// SIMATIC STEP 7 (V5.x) project aplicaciopnes
// CPU: CPU 314C-2 DP
// CPU: CPU 314C-2 DP
// CPU: CPU 314C-2 DP
// CPU: CPU 314C-2 DP
// CPU: CPU 314C-2 DP
// CPU: CPU 314C-2 DP
// CPU: CPU 314C-2 DP
// station: Hardware
// station: secuencial
// station: P_ADR_BUS
// station: Hardware
// station: motores secuenciales
// station: P_ADR_BUS
// station: Hardware
// station: mot sec original
// station: P_ADR_BUS
// station: Hardware
// station: agitador con agua
// station: P_ADR_BUS
// station: Hardware
// station: bombas con una lampara
// station: P_ADR_BUS
// station: Hardware
// station: funciones
// station: P_ADR_BUS
// station: Hardware
// station: tres tanques llenado sec
// station: P_ADR_BUS
// program: Programa S7(1)
// program: Programa S7(2)
// program: Programa S7(3)
// program: Programa S7(5)
// program: Programa S7(6)
// program: Programa S7(7)
// program: Programa S7(8)

SYMBOL_TABLE
"arranque"	I 124.0	BOOL
"paro"	I 124.1	BOOL
"L1"	Q 124.0	BOOL
"L2"	Q 124.1	BOOL
"L3"	Q 124.2	BOOL
END_SYMBOL_TABLE

ORGANIZATION_BLOCK OB 1
TITLE = "Main Program Sweep (Cycle)"
VERSION : 0.1
VAR_TEMP
  OB1_EV_CLASS : BYTE ;	//Bits 0-3 = 1 (Coming event), Bits 4-7 = 1 (Event class 1)
  OB1_SCAN_1 : BYTE ;	//1 (Cold restart scan 1 of OB 1), 3 (Scan 2-n of OB 1)
  OB1_PRIORITY : BYTE ;	//Priority of OB Execution
  OB1_OB_NUMBR : BYTE ;	//1 (Organization block 1, OB1)
  OB1_RESERVED_1 : BYTE ;	//Reserved for system
  OB1_RESERVED_2 : BYTE ;	//Reserved for system
  OB1_PREV_CYCLE : INT ;	//Cycle time of previous OB1 scan (milliseconds)
  OB1_MIN_CYCLE : INT ;	//Minimum cycle time of OB1 (milliseconds)
  OB1_MAX_CYCLE : INT ;	//Maximum cycle time of OB1 (milliseconds)
  OB1_DATE_TIME : DATE_AND_TIME ;	//Date and time OB1 started
END_VAR
BEGIN
NETWORK
TITLE =
      A(;
      A     "arranque";
      FN    M 0.1;
      S     M 0.0;
      A     "paro";
      R     M 0.0;
      A     M 0.0;
      );
      A     M 0.5;
      =     Q 124.5;
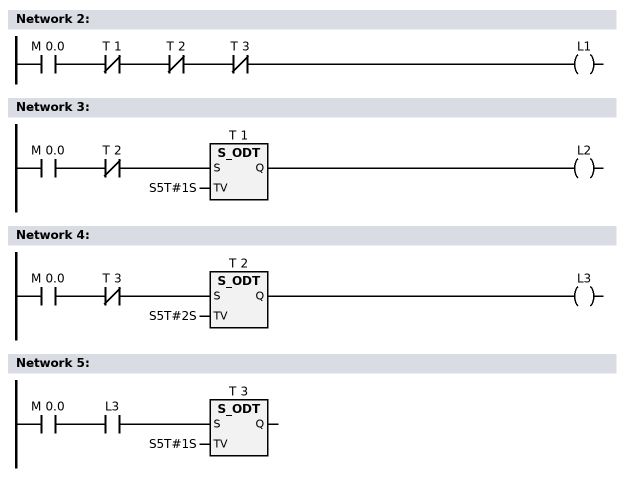
NETWORK
TITLE =
      A     M 0.0;
      AN    T 1;
      AN    T 2;
      AN    T 3;
      =     "L1";
NETWORK
TITLE =
      A     M 0.0;
      AN    T 2;
      L     S5T#1S;
      SD    T 1;
      NOP   0;
      NOP   0;
      NOP   0;
      A     T 1;
      =     "L2";
NETWORK
TITLE =
      A     M 0.0;
      AN    T 3;
      L     S5T#2S;
      SD    T 2;
      NOP   0;
      NOP   0;
      NOP   0;
      A     T 2;
      =     "L3";
NETWORK
TITLE =
      A     M 0.0;
      A     "L3";
      L     S5T#1S;
      SD    T 3;
      NOP   0;
      NOP   0;
      NOP   0;
      NOP   0;
END_ORGANIZATION_BLOCK

SYMBOL_TABLE
"arranque"	I 124.0	BOOL
"paro"	I 124.1	BOOL
"motor 1"	Q 124.0	BOOL
"motor 2"	Q 124.1	BOOL
"motor 3"	Q 124.2	BOOL
"lampara v1"	Q 124.3	BOOL
"lampara v2"	Q 124.4	BOOL
"lampara v3"	Q 124.5	BOOL
"lampara r1"	Q 124.6	BOOL
"lampara r2"	Q 124.7	BOOL
"lampara r3"	Q 125.0	BOOL
END_SYMBOL_TABLE

ORGANIZATION_BLOCK OB 1
TITLE = "Main Program Sweep (Cycle)"
VERSION : 0.1
VAR_TEMP
  OB1_EV_CLASS : BYTE ;	//Bits 0-3 = 1 (Coming event), Bits 4-7 = 1 (Event class 1)
  OB1_SCAN_1 : BYTE ;	//1 (Cold restart scan 1 of OB 1), 3 (Scan 2-n of OB 1)
  OB1_PRIORITY : BYTE ;	//Priority of OB Execution
  OB1_OB_NUMBR : BYTE ;	//1 (Organization block 1, OB1)
  OB1_RESERVED_1 : BYTE ;	//Reserved for system
  OB1_RESERVED_2 : BYTE ;	//Reserved for system
  OB1_PREV_CYCLE : INT ;	//Cycle time of previous OB1 scan (milliseconds)
  OB1_MIN_CYCLE : INT ;	//Minimum cycle time of OB1 (milliseconds)
  OB1_MAX_CYCLE : INT ;	//Maximum cycle time of OB1 (milliseconds)
  OB1_DATE_TIME : DATE_AND_TIME ;	//Date and time OB1 started
END_VAR
BEGIN
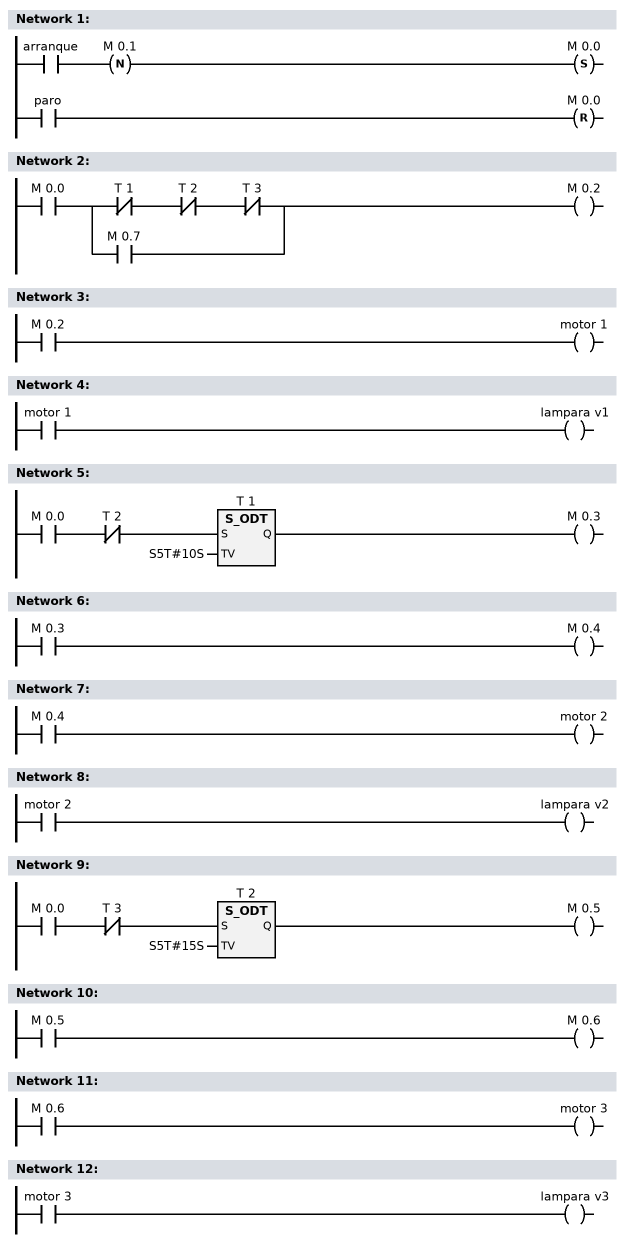
NETWORK
TITLE =
      A     "arranque";
      FN    M 0.1;
      S     M 0.0;
      A     "paro";
      R     M 0.0;
      NOP   0;
NETWORK
TITLE =
      A     M 0.0;
      A(;
      AN    T 1;
      AN    T 2;
      AN    T 3;
      O     M 0.7;
      );
      =     M 0.2;
NETWORK
TITLE =
      A     M 0.2;
      =     "motor 1";
NETWORK
TITLE =
      A     "motor 1";
      =     "lampara v1";
NETWORK
TITLE =
      A     M 0.0;
      AN    T 2;
      L     S5T#10S;
      SD    T 1;
      NOP   0;
      NOP   0;
      NOP   0;
      A     T 1;
      =     M 0.3;
NETWORK
TITLE =
      A     M 0.3;
      =     M 0.4;
NETWORK
TITLE =
      A     M 0.4;
      =     "motor 2";
NETWORK
TITLE =
      A     "motor 2";
      =     "lampara v2";
NETWORK
TITLE =
      A     M 0.0;
      AN    T 3;
      L     S5T#15S;
      SD    T 2;
      NOP   0;
      NOP   0;
      NOP   0;
      A     T 2;
      =     M 0.5;
NETWORK
TITLE =
      A     M 0.5;
      =     M 0.6;
NETWORK
TITLE =
      A     M 0.6;
      =     "motor 3";
NETWORK
TITLE =
      A     "motor 3";
      =     "lampara v3";
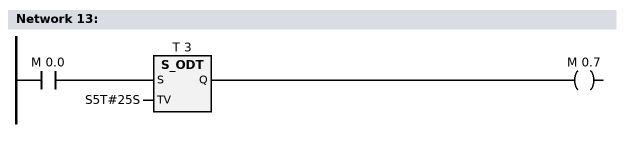
NETWORK
TITLE =
      A     M 0.0;
      L     S5T#25S;
      SD    T 3;
      NOP   0;
      NOP   0;
      NOP   0;
      A     T 3;
      =     M 0.7;
END_ORGANIZATION_BLOCK

SYMBOL_TABLE
"sensor temp baja"	I 124.0	BOOL
"sensor temp alta"	I 124.1	BOOL
"sensor press baja"	I 124.2	BOOL
"sensor press alta"	I 124.3	BOOL
"temperatura normal"	M 0.0	BOOL
"presion normal"	M 0.1	BOOL
"valvula seguridad"	Q 124.0	BOOL
"calentador"	Q 124.1	BOOL
"enfriador"	Q 124.2	BOOL
"agitador"	Q 124.3	BOOL
END_SYMBOL_TABLE

ORGANIZATION_BLOCK OB 1
TITLE = "Main Program Sweep (Cycle)"
VERSION : 0.1
VAR_TEMP
  OB1_EV_CLASS : BYTE ;	//Bits 0-3 = 1 (Coming event), Bits 4-7 = 1 (Event class 1)
  OB1_SCAN_1 : BYTE ;	//1 (Cold restart scan 1 of OB 1), 3 (Scan 2-n of OB 1)
  OB1_PRIORITY : BYTE ;	//Priority of OB Execution
  OB1_OB_NUMBR : BYTE ;	//1 (Organization block 1, OB1)
  OB1_RESERVED_1 : BYTE ;	//Reserved for system
  OB1_RESERVED_2 : BYTE ;	//Reserved for system
  OB1_PREV_CYCLE : INT ;	//Cycle time of previous OB1 scan (milliseconds)
  OB1_MIN_CYCLE : INT ;	//Minimum cycle time of OB1 (milliseconds)
  OB1_MAX_CYCLE : INT ;	//Maximum cycle time of OB1 (milliseconds)
  OB1_DATE_TIME : DATE_AND_TIME ;	//Date and time OB1 started
END_VAR
BEGIN
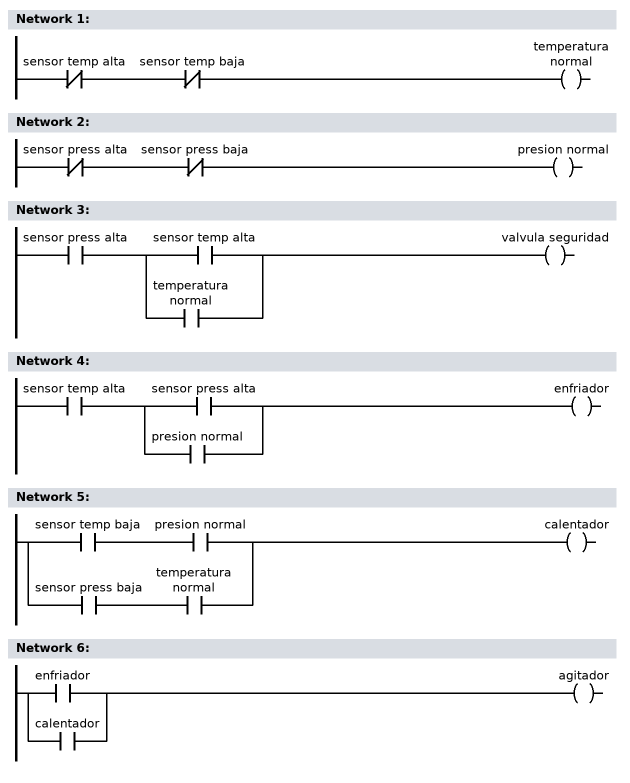
NETWORK
TITLE =
//temperatura normal
      AN    "sensor temp alta";
      AN    "sensor temp baja";
      =     "temperatura normal";
NETWORK
TITLE =
//presion normal
      AN    "sensor press alta";
      AN    "sensor press baja";
      =     "presion normal";
NETWORK
TITLE =
//activacion de valvula de seguridad
      A     "sensor press alta";
      A(;
      O     "sensor temp alta";
      O     "temperatura normal";
      );
      =     "valvula seguridad";
NETWORK
TITLE =
//activacion de enfriador
      A     "sensor temp alta";
      A(;
      O     "sensor press alta";
      O     "presion normal";
      );
      =     "enfriador";
NETWORK
TITLE =
//activacion de calentador
      A     "sensor temp baja";
      A     "presion normal";
      O;
      A     "sensor press baja";
      A     "temperatura normal";
      =     "calentador";
NETWORK
TITLE =
//activacion de agitador
      O     "enfriador";
      O     "calentador";
      =     "agitador";
END_ORGANIZATION_BLOCK

SYMBOL_TABLE
"marcha 1"	I 124.0	BOOL
"marcha 2"	I 124.1	BOOL
"marcha 3"	I 124.2	BOOL
"paro 1"	I 124.3	BOOL
"paro 2"	I 124.4	BOOL
"paro 3"	I 124.5	BOOL
"marcha"	I 124.6	BOOL
"parada"	I 124.7	BOOL
"lampara h"	Q 124.0	BOOL
"bomba 1"	Q 124.1	BOOL
"bomba 2"	Q 124.2	BOOL
"bomba 3"	Q 124.3	BOOL
END_SYMBOL_TABLE

ORGANIZATION_BLOCK OB 1
TITLE = "Main Program Sweep (Cycle)"
VERSION : 0.1
VAR_TEMP
  OB1_EV_CLASS : BYTE ;	//Bits 0-3 = 1 (Coming event), Bits 4-7 = 1 (Event class 1)
  OB1_SCAN_1 : BYTE ;	//1 (Cold restart scan 1 of OB 1), 3 (Scan 2-n of OB 1)
  OB1_PRIORITY : BYTE ;	//Priority of OB Execution
  OB1_OB_NUMBR : BYTE ;	//1 (Organization block 1, OB1)
  OB1_RESERVED_1 : BYTE ;	//Reserved for system
  OB1_RESERVED_2 : BYTE ;	//Reserved for system
  OB1_PREV_CYCLE : INT ;	//Cycle time of previous OB1 scan (milliseconds)
  OB1_MIN_CYCLE : INT ;	//Minimum cycle time of OB1 (milliseconds)
  OB1_MAX_CYCLE : INT ;	//Maximum cycle time of OB1 (milliseconds)
  OB1_DATE_TIME : DATE_AND_TIME ;	//Date and time OB1 started
END_VAR
BEGIN
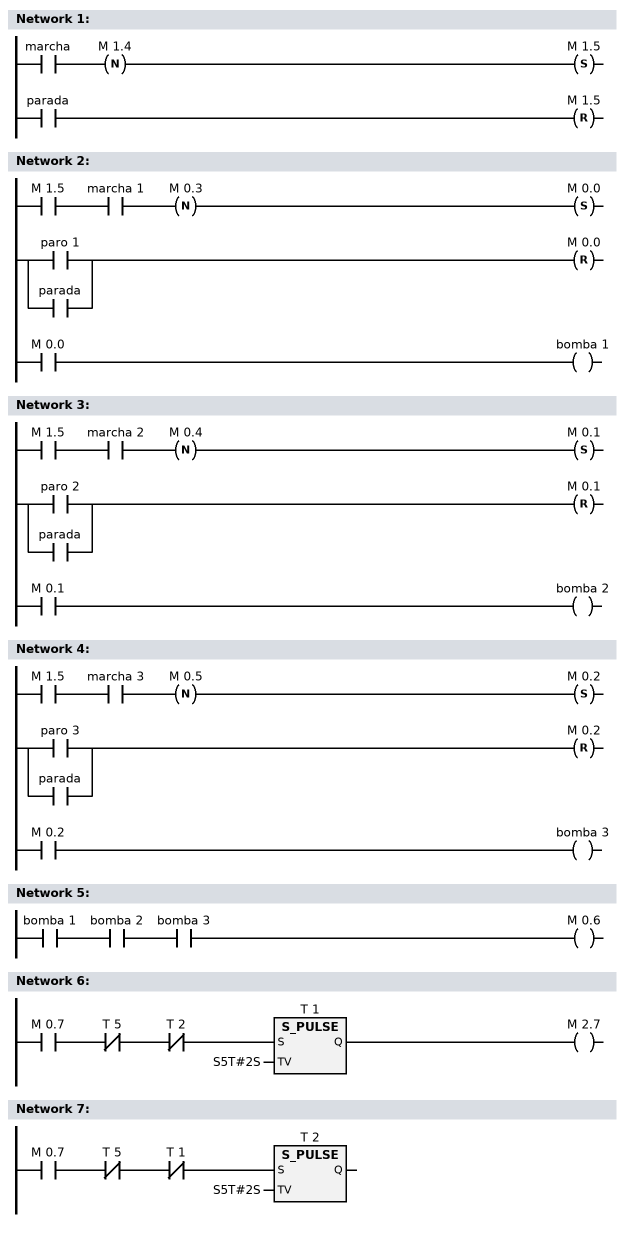
NETWORK
TITLE =
      A     "marcha";
      FN    M 1.4;
      S     M 1.5;
      A     "parada";
      R     M 1.5;
      NOP   0;
NETWORK
TITLE =
      A     M 1.5;
      A     "marcha 1";
      FN    M 0.3;
      S     M 0.0;
      A(;
      O     "paro 1";
      O     "parada";
      );
      R     M 0.0;
      A     M 0.0;
      =     "bomba 1";
NETWORK
TITLE =
      A     M 1.5;
      A     "marcha 2";
      FN    M 0.4;
      S     M 0.1;
      A(;
      O     "paro 2";
      O     "parada";
      );
      R     M 0.1;
      A     M 0.1;
      =     "bomba 2";
NETWORK
TITLE =
      A     M 1.5;
      A     "marcha 3";
      FN    M 0.5;
      S     M 0.2;
      A(;
      O     "paro 3";
      O     "parada";
      );
      R     M 0.2;
      A     M 0.2;
      =     "bomba 3";
NETWORK
TITLE =
      A     "bomba 1";
      A     "bomba 2";
      A     "bomba 3";
      =     M 0.6;
NETWORK
TITLE =
      A     M 0.7;
      AN    T 5;
      AN    T 2;
      L     S5T#2S;
      SP    T 1;
      NOP   0;
      NOP   0;
      NOP   0;
      A     T 1;
      =     M 2.7;
NETWORK
TITLE =
      A     M 0.7;
      AN    T 5;
      AN    T 1;
      L     S5T#2S;
      SP    T 2;
      NOP   0;
      NOP   0;
      NOP   0;
      NOP   0;
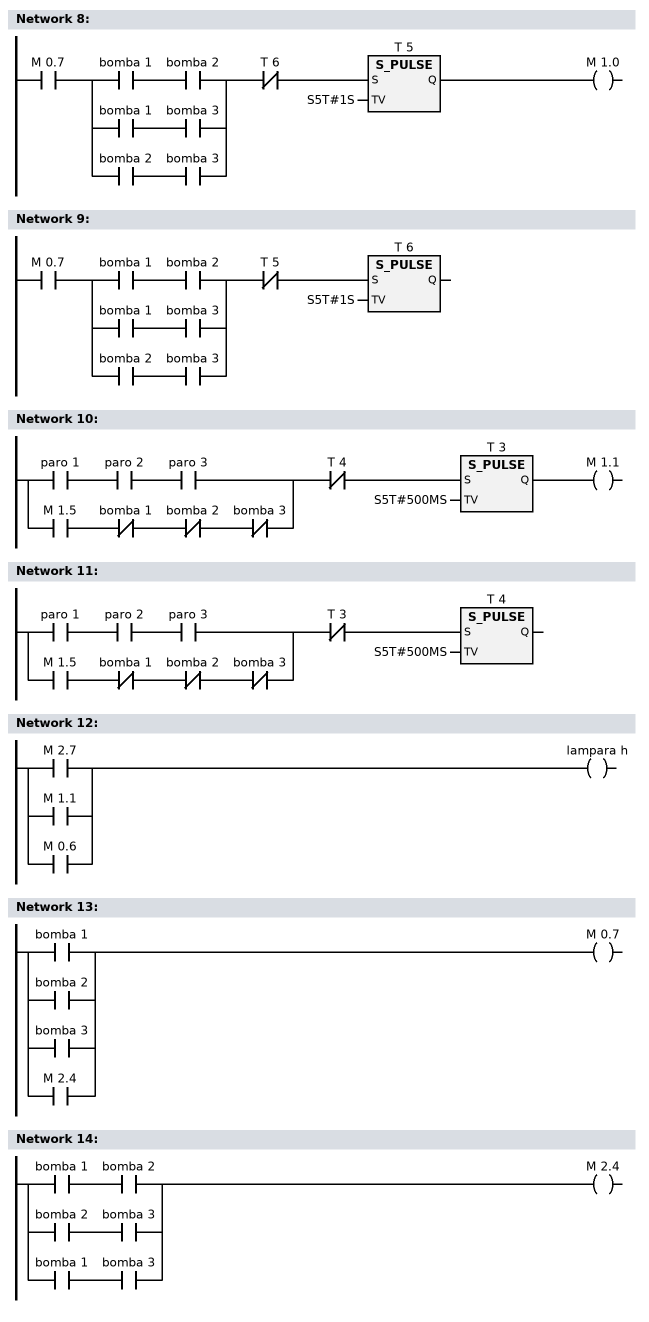
NETWORK
TITLE =
      A     M 0.7;
      A(;
      A     "bomba 1";
      A     "bomba 2";
      O;
      A     "bomba 1";
      A     "bomba 3";
      O;
      A     "bomba 2";
      A     "bomba 3";
      );
      AN    T 6;
      L     S5T#1S;
      SP    T 5;
      NOP   0;
      NOP   0;
      NOP   0;
      A     T 5;
      =     M 1.0;
NETWORK
TITLE =
      A     M 0.7;
      A(;
      A     "bomba 1";
      A     "bomba 2";
      O;
      A     "bomba 1";
      A     "bomba 3";
      O;
      A     "bomba 2";
      A     "bomba 3";
      );
      AN    T 5;
      L     S5T#1S;
      SP    T 6;
      NOP   0;
      NOP   0;
      NOP   0;
      NOP   0;
NETWORK
TITLE =
      A(;
      A     "paro 1";
      A     "paro 2";
      A     "paro 3";
      O;
      A     M 1.5;
      AN    "bomba 1";
      AN    "bomba 2";
      AN    "bomba 3";
      );
      AN    T 4;
      L     S5T#500MS;
      SP    T 3;
      NOP   0;
      NOP   0;
      NOP   0;
      A     T 3;
      =     M 1.1;
NETWORK
TITLE =
      A(;
      A     "paro 1";
      A     "paro 2";
      A     "paro 3";
      O;
      A     M 1.5;
      AN    "bomba 1";
      AN    "bomba 2";
      AN    "bomba 3";
      );
      AN    T 3;
      L     S5T#500MS;
      SP    T 4;
      NOP   0;
      NOP   0;
      NOP   0;
      NOP   0;
NETWORK
TITLE =
      O     M 2.7;
      O     M 1.1;
      O     M 0.6;
      =     "lampara h";
NETWORK
TITLE =
      O     "bomba 1";
      O     "bomba 2";
      O     "bomba 3";
      O     M 2.4;
      =     M 0.7;
NETWORK
TITLE =
      A     "bomba 1";
      A     "bomba 2";
      O;
      A     "bomba 2";
      A     "bomba 3";
      O;
      A     "bomba 1";
      A     "bomba 3";
      =     M 2.4;
END_ORGANIZATION_BLOCK

SYMBOL_TABLE
"generador de pulsos"	FC 1	FC 1
END_SYMBOL_TABLE

FUNCTION "generador de pulsos" : VOID	// FC 1
VERSION : 0.1
VAR_INPUT
  on_off : BOOL ;
  timerA : TIMER ;
  timerB : TIMER ;
  tiempo : S5TIME ;
END_VAR
VAR_OUTPUT
  pulsos : BOOL ;
END_VAR
BEGIN
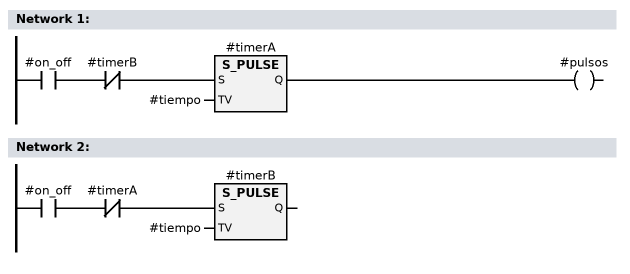
NETWORK
TITLE =
      A     #on_off;
      AN    #timerB;
      L     #tiempo;
      SP    #timerA;
      NOP   0;
      NOP   0;
      NOP   0;
      A     #timerA;
      =     #pulsos;
NETWORK
TITLE =
      A     #on_off;
      AN    #timerA;
      L     #tiempo;
      SP    #timerB;
      NOP   0;
      NOP   0;
      NOP   0;
      NOP   0;
END_FUNCTION

ORGANIZATION_BLOCK OB 1
TITLE = "Main Program Sweep (Cycle)"
VERSION : 0.1
VAR_TEMP
  OB1_EV_CLASS : BYTE ;	//Bits 0-3 = 1 (Coming event), Bits 4-7 = 1 (Event class 1)
  OB1_SCAN_1 : BYTE ;	//1 (Cold restart scan 1 of OB 1), 3 (Scan 2-n of OB 1)
  OB1_PRIORITY : BYTE ;	//Priority of OB Execution
  OB1_OB_NUMBR : BYTE ;	//1 (Organization block 1, OB1)
  OB1_RESERVED_1 : BYTE ;	//Reserved for system
  OB1_RESERVED_2 : BYTE ;	//Reserved for system
  OB1_PREV_CYCLE : INT ;	//Cycle time of previous OB1 scan (milliseconds)
  OB1_MIN_CYCLE : INT ;	//Minimum cycle time of OB1 (milliseconds)
  OB1_MAX_CYCLE : INT ;	//Maximum cycle time of OB1 (milliseconds)
  OB1_DATE_TIME : DATE_AND_TIME ;	//Date and time OB1 started
END_VAR
BEGIN
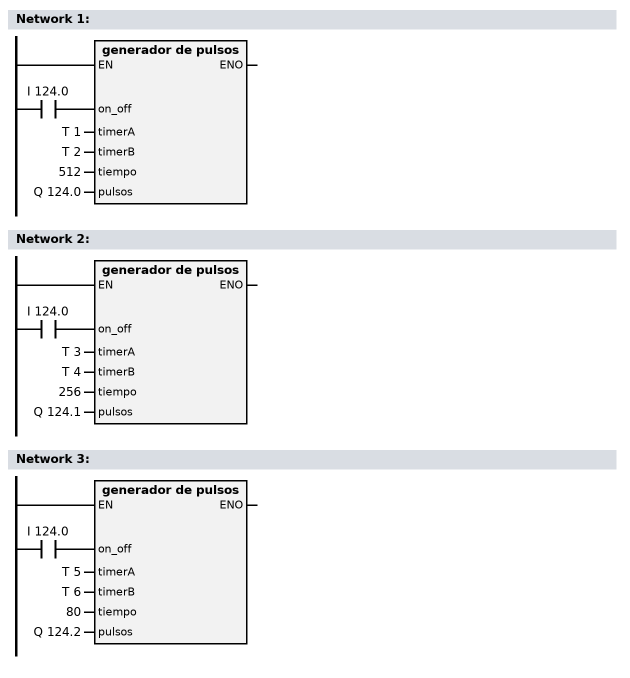
NETWORK
TITLE =
      A     I 124.0;
      =     L 20.0;
      BLD   103;
      CALL  "generador de pulsos" (
           on_off                   := L 20.0,
           timerA                   := T 1,
           timerB                   := T 2,
           tiempo                   := 512,
           pulsos                   := Q 124.0);
      NOP   0;
NETWORK
TITLE =
      A     I 124.0;
      =     L 20.0;
      BLD   103;
      CALL  "generador de pulsos" (
           on_off                   := L 20.0,
           timerA                   := T 3,
           timerB                   := T 4,
           tiempo                   := 256,
           pulsos                   := Q 124.1);
      NOP   0;
NETWORK
TITLE =
      A     I 124.0;
      =     L 20.0;
      BLD   103;
      CALL  "generador de pulsos" (
           on_off                   := L 20.0,
           timerA                   := T 5,
           timerB                   := T 6,
           tiempo                   := 80,
           pulsos                   := Q 124.2);
      NOP   0;
END_ORGANIZATION_BLOCK

SYMBOL_TABLE
"paro"	I 124.0	BOOL
"marcha"	I 124.1	BOOL
"sensor na 1"	I 124.2	BOOL
"sensor na 2"	I 124.3	BOOL
"sensor na 3"	I 124.4	BOOL
"sensor nc 1"	I 124.5	BOOL
"sensor nc 2"	I 124.6	BOOL
"sensor nc 3"	I 124.7	BOOL
"tanque y1"	Q 124.0	BOOL
"tanque y2"	Q 124.1	BOOL
"tanque y3"	Q 124.2	BOOL
END_SYMBOL_TABLE

ORGANIZATION_BLOCK OB 1
TITLE = "Main Program Sweep (Cycle)"
VERSION : 0.1
VAR_TEMP
  OB1_EV_CLASS : BYTE ;	//Bits 0-3 = 1 (Coming event), Bits 4-7 = 1 (Event class 1)
  OB1_SCAN_1 : BYTE ;	//1 (Cold restart scan 1 of OB 1), 3 (Scan 2-n of OB 1)
  OB1_PRIORITY : BYTE ;	//Priority of OB Execution
  OB1_OB_NUMBR : BYTE ;	//1 (Organization block 1, OB1)
  OB1_RESERVED_1 : BYTE ;	//Reserved for system
  OB1_RESERVED_2 : BYTE ;	//Reserved for system
  OB1_PREV_CYCLE : INT ;	//Cycle time of previous OB1 scan (milliseconds)
  OB1_MIN_CYCLE : INT ;	//Minimum cycle time of OB1 (milliseconds)
  OB1_MAX_CYCLE : INT ;	//Maximum cycle time of OB1 (milliseconds)
  OB1_DATE_TIME : DATE_AND_TIME ;	//Date and time OB1 started
END_VAR
BEGIN
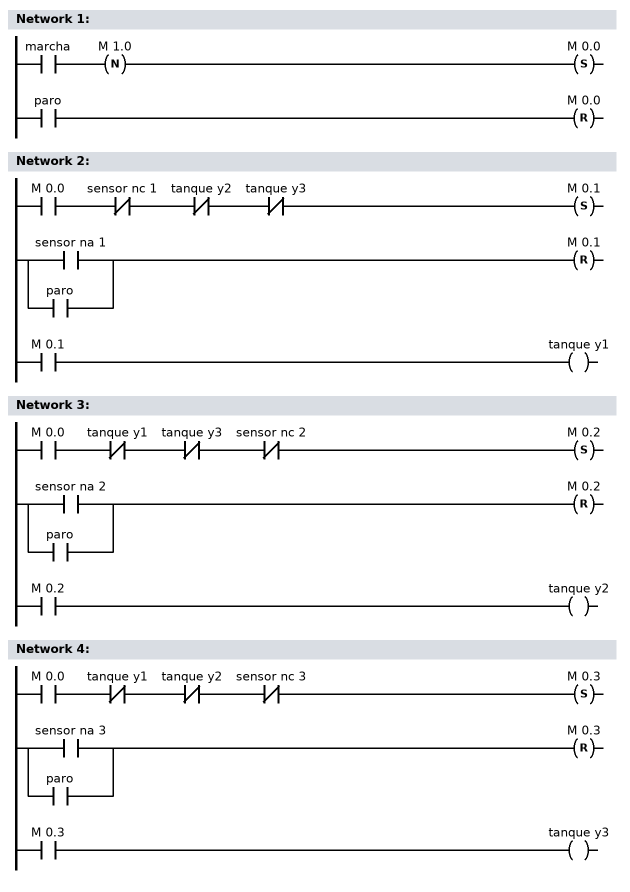
NETWORK
TITLE =
      A     "marcha";
      FN    M 1.0;
      S     M 0.0;
      A     "paro";
      R     M 0.0;
      NOP   0;
NETWORK
TITLE =
      A     M 0.0;
      AN    "sensor nc 1";
      AN    "tanque y2";
      AN    "tanque y3";
      S     M 0.1;
      A(;
      O     "sensor na 1";
      O     "paro";
      );
      R     M 0.1;
      A     M 0.1;
      =     "tanque y1";
NETWORK
TITLE =
      A     M 0.0;
      AN    "tanque y1";
      AN    "tanque y3";
      AN    "sensor nc 2";
      S     M 0.2;
      A(;
      O     "sensor na 2";
      O     "paro";
      );
      R     M 0.2;
      A     M 0.2;
      =     "tanque y2";
NETWORK
TITLE =
      A     M 0.0;
      AN    "tanque y1";
      AN    "tanque y2";
      AN    "sensor nc 3";
      S     M 0.3;
      A(;
      O     "sensor na 3";
      O     "paro";
      );
      R     M 0.3;
      A     M 0.3;
      =     "tanque y3";
END_ORGANIZATION_BLOCK

SYMBOL_TABLE
"arranque"	I 124.0	BOOL
"paro"	I 124.1	BOOL
""	I 124.2	BOOL
END_SYMBOL_TABLE
